// TwinCAT 3 PLC project Untitled1
// ProgramVersion: 3.1.4024.0
// libraries:
//   Tc2_Standard, * (Beckhoff Automation GmbH)
//   Tc2_System, * (Beckhoff Automation GmbH)
//   Tc2_TcpIp, * (Beckhoff Automation GmbH)
//   Tc3_Module, * (Beckhoff Automation GmbH)
// project tree:
//   / PlcTask.TcTTO
//   POUs/ FB_Systems.TcPOU, FB_TcpClient.TcPOU, I_Tcp.TcIO, MAIN.TcPOU, ST_ServerResponse.TcDUT
// real-time tasks:
//   TASK PlcTask: cycle T#10ms, priority 20, ADS port 350

CONFIGURATION Untitled1
    RESOURCE PLC ON TwinCAT3
        TASK PlcTask(INTERVAL := T#10ms, PRIORITY := 20);
        PROGRAM MAIN WITH PlcTask : MAIN;
    END_RESOURCE
END_CONFIGURATION

// ---- POUs/ST_ServerResponse.TcDUT
TYPE ST_ServerResponse :
STRUCT
	nStatus     : INT;
    fValue      : REAL;
    nErrorCode  : INT;
END_STRUCT
END_TYPE

// ---- POUs/I_Tcp.TcIO
INTERFACE I_Tcp

PROPERTY IsConnected : bool
GET
END_GET
END_PROPERTY

METHOD M_Connect
VAR_INPUT
	sIP   : STRING(15);
    nPort : UINT;
END_VAR
END_METHOD

METHOD M_Disconnect
VAR_INPUT
END_VAR
END_METHOD

METHOD M_Send
VAR_INPUT
	pData : POINTER TO BYTE; 
    nSize : UDINT;
END_VAR
END_METHOD

END_INTERFACE

// ---- POUs/MAIN.TcPOU
PROGRAM MAIN
VAR
	Hethong2 : FB_Systems;
END_VAR

Hethong2();

END_PROGRAM

// ---- POUs/FB_Systems.TcPOU
FUNCTION_BLOCK FB_Systems
VAR_INPUT
END_VAR
VAR_OUTPUT
END_VAR
VAR
	ClientTCP : FB_TcpClient;
    
    bKetNoi   : BOOL;
    bGuiData  : BOOL;

    sMessage  : STRING := 'Hello Server OOP';
END_VAR

ClientTCP.M_Execute();

IF bKetNoi AND NOT ClientTCP.IsConnected THEN
    ClientTCP.M_Connect(sIP := '192.168.1.100', nPort := 502); 
    bKetNoi := FALSE; 
END_IF

IF bGuiData AND ClientTCP.IsConnected THEN
    ClientTCP.M_Send(
        pData := ADR(sMessage), 
        nSize := INT_TO_UDINT(LEN(sMessage))
    );
    bGuiData := FALSE;
END_IF

END_FUNCTION_BLOCK

// ---- POUs/FB_TcpClient.TcPOU
FUNCTION_BLOCK FB_TcpClient IMPLEMENTS I_Tcp
VAR_INPUT
END_VAR
VAR_OUTPUT
END_VAR
VAR

    fbConnect       : FB_SocketConnect;
    fbClose         : FB_SocketClose;
    fbSend          : FB_SocketSend;
    fbReceive       : FB_SocketReceive;
    
    hSocket         : T_HSOCKET; 
    _bConnected     : BOOL;
    nState          : INT := 0;  
    

    arrRxBuffer     : ARRAY[0..255] OF BYTE;
    nBytesReceived  : UDINT;
	stRxData        : ST_ServerResponse;

    bCmdConnect     : BOOL;
    bCmdDisconnect  : BOOL;
    bCmdSend        : BOOL;
    
    sIP_Address     : STRING(15);
    nTargetPort     : UINT;
    
    pSendData       : POINTER TO BYTE;
    nSendSize       : UDINT;
END_VAR

{warning 'add property implementation'}
PROPERTY IsConnected : BOOL
GET
IsConnected := _bConnected;
END_GET
END_PROPERTY

{warning 'add method implementation '}
METHOD M_Connect
VAR_INPUT
	sIP	: STRING(15);
	nPort	: UINT;
END_VAR
sIP_Address := sIP;
nTargetPort := nPort;

bCmdConnect := TRUE;
bCmdDisconnect := FALSE;
END_METHOD

{warning 'add method implementation '}
METHOD M_Disconnect
bCmdDisconnect := TRUE;
bCmdConnect := FALSE;
END_METHOD

METHOD M_Execute
VAR_INPUT
END_VAR
CASE nState OF
    0:
        IF bCmdConnect THEN
            fbConnect(
                sSrvNetId   := '', 
                sRemoteHost := sIP_Address, 
                nRemotePort := nTargetPort, 
                bExecute    := TRUE, 
                tTimeout    := T#3S
            );
            nState := 10;
        END_IF

    10:
        fbConnect(bExecute := FALSE);
        IF NOT fbConnect.bBusy THEN
            IF NOT fbConnect.bError THEN
                hSocket := fbConnect.hSocket;
                _bConnected := TRUE;
                nState := 20;
                nState := 99;
            END_IF
        END_IF

    20: 
        fbReceive(
            hSocket     := hSocket,
            cbLen       := SIZEOF(arrRxBuffer),
            pDest       := ADR(arrRxBuffer),
            bExecute    := TRUE,
            tTimeout    := T#1S
        );
        IF NOT fbReceive.bBusy THEN
            IF NOT fbReceive.bError AND fbReceive.nRecBytes > 0 THEN
                nBytesReceived := fbReceive.nRecBytes;
                MEMCPY(ADR(stRxData), ADR(arrRxBuffer), SIZEOF(stRxData));
            END_IF
            fbReceive(bExecute := FALSE);
        END_IF

        IF bCmdDisconnect THEN
            _bConnected := FALSE;
            nState := 30;
        END_IF

    30:
        fbClose(
            hSocket  := hSocket,
            bExecute := TRUE,
            tTimeout := T#1S
        );
        IF NOT fbClose.bBusy THEN
            fbClose(bExecute := FALSE);
            nState := 0; 
        END_IF
        
    99: 
        _bConnected := FALSE;
END_CASE
END_METHOD

{warning 'add method implementation '}
METHOD M_Send
VAR_INPUT
	pData	: POINTER TO BYTE;
	nSize	: UDINT;
END_VAR
pSendData := pData;
nSendSize := nSize;

bCmdSend := TRUE;
END_METHOD

END_FUNCTION_BLOCK
